FUNCTION_BLOCK RampUp
VAR_INPUT
	IN: BOOL;
	RampUpTime: TIME;
	Ramp_lowerLimit: REAL;
	Ramp_upperLimit: REAL;
	PLC_CYCLE_TIME_ms: REAL;
END_VAR
VAR_IN_OUT
	output: REAL;
END_VAR
VAR_OUTPUT
	InProgress: BOOL;	
END_VAR
VAR
	rampUp: REAL;
	x: REAL;
	init: BOOL;
END_VAR


	IF IN AND (RampUpTime > T#0S) AND (PLC_CYCLE_TIME_ms > 0) THEN
		IF NOT init THEN
			init	:=	TRUE;
			InProgress	:=	TRUE;
			rampUp	:=	TIME_TO_REAL(RampUpTime);		
			x		:=	PLC_CYCLE_TIME_ms / rampUp;
			x		:=	(Ramp_upperLimit - Ramp_lowerLimit) * x;	
		END_IF
		
		IF (output < Ramp_upperLimit) AND (InProgress) THEN
			output		:=	output + x;
		ELSE
			output		:=	Ramp_upperLimit;
			InProgress	:=	FALSE;
		END_IF
		
	ELSE
		InProgress 	:=	FALSE;	
		init		:=	FALSE;
	END_IF

END_FUNCTION_BLOCK

(* stored: Version 1.1.0.1, ProductVersion 3.1.4024.13
   POU RampUp: Id {dd705717-ae7c-44f5-9b09-3e860dfa96d6}, SpecialFunc None *)
